Fanuc TP program (LS listing): S103_PK_T13N50.LS

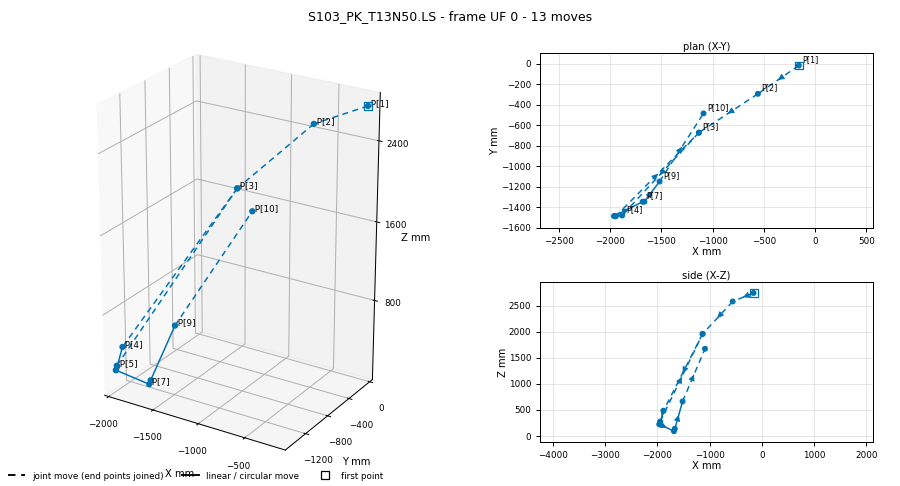
[picture p0: tool path of S103_PK_T13N50.LS in frame UF 0, 13 of 15 moves have a stored position in this frame; points joined in program order, loops and branches not executed]
/PROG  S103_PK_T13N50
/ATTR
OWNER		= MNEDITOR;
COMMENT		= "TL PCK TYP1 N50";
PROG_SIZE	= 4491;
CREATE		= DATE 21-06-09  TIME 06:41:38;
MODIFIED	= DATE 21-06-09  TIME 12:42:18;
FILE_NAME	= S103_PK_;
VERSION		= 0;
LINE_COUNT	= 155;
MEMORY_SIZE	= 4911;
PROTECT		= READ_WRITE;
STORAGE		= SHADOW;
TCD:  STACK_SIZE	= 0,
      TASK_PRIORITY	= 50,
      TIME_SLICE	= 0,
      BUSY_LAMP_OFF	= 0,
      ABORT_REQUEST	= 0,
      PAUSE_REQUEST	= 0;
DEFAULT_GROUP	= 1,*,*,*,*;
CONTROL_CODE	= 00000000 00000000;
/APPL
  HANDLING : TRUE ;
/MN
   1:  !******************************** ;
   2:  ! PATH - PK TOOL FROM N1=STA 70 ;
   3:  !******************************** ;
   4:  !* Robot ID: XXXXXR02B1 ;
   5:  !*    F-19XXXX ;
   6:  !* Line: XXXXXXXX ;
   7:  !* Platform: XX ;
   8:  !* Tool ID: TOOL xx ;
   9:  !* Program: S001_PK_TxxN3_R02 ;
  10:  !* Application: TOOL PICK ;
  11:  !******************************** ;
  12:  ! Author- Esys Automation ;
  13:  !******************************** ;
  14:   ;
  15:  !++++++++++++++++++++++++++++++++ ;
  16:  !ASSIGN PROGRAM PATH VALUES ;
  17:  !-------------------------------- ;
  18:  !Set ATI Tool and World UFrame ;
  19:  UTOOL_NUM=14 ;
  20:  UFRAME_NUM=0 ;
  21:  !++++++++++++++++++++++++++++++++ ;
  22:   ;
  23:  !******************************** ;
  24:  !BEGINNING OF PROGRAM PATH ;
  25:  !MOVE TO NEST 1 TOOL PICK ;
  26:  !******************************** ;
  27:   ;
  28:  !-------------------------------- ;
  29:  LBL[10:MOVE TO TL PICK] ;
  30:   ;
  31:  SET SEGMENT(52) ;
  32:  !SEG(52), Approach Tool Pick ;
  33:   ;
  34:   ;
  35:J P[1] 100% CNT100    ;
  36:J P[2] 100% CNT100    ;
  37:J P[3] 100% CNT100    ;
  38:J P[4] 100% CNT100    ;
  39:   ;
  40:L P[5] 200mm/sec FINE    ;
  41:   ;
  42:L P[6:Pick Tool] 50mm/sec FINE    ;
  43:   ;
  44:  !-------------------------------- ;
  45:  LBL[20:LATCH TOOL] ;
  46:  LATCH TOOL    ;
  47:   ;
  48:  !Add MH Ethernet Device from ;
  49:  !I/O Ethernet table ;
  50:  !which tool has ;
  51:   ;
  52:  !ADD DEVICE ONLINE CALLS ;
  53:  !WITHOUT STATUS CHECK ARG ;
  54:  !FOR ALL EOAT DEVICES ;
  55:  !CALL EN_ONLN(x,y) ;
  56:  !x = EOAT ENET Node # ;
  57:  !y = wait time ;
  58:  CALL EN_ONLN(31,5) ;
  59:  CALL EN_AROFF(31) ;
  60:   ;
  61:  !If TL LCH Pass, Return Home ;
  62:  !If TL LCH Fail, Unlatch TL, ;
  63:  !  MHFault, and Return Home ;
  64:  IF R[170]=1,JMP LBL[30] ;
  65:   ;
  66:  SELECT R[168]=6,JMP LBL[80] ;
  67:         ELSE,JMP LBL[99] ;
  68:   ;
  69:  !-------------------------------- ;
  70:  LBL[30:TOOL CHECK] ;
  71:   ;
  72:  ! Check if Tool Match with PLC ;
  73:  CALL TL_CHK_KM(R[156]) ;
  74:   ;
  75:  !If TL CHK Pass, Return Home ;
  76:  !If TL CHK Fail, Unlatch Tool, ;
  77:  !  MHFault, and Return Home ;
  78:  IF R[170]=1,JMP LBL[40] ;
  79:  IF R[170]=0,JMP LBL[905] ;
  80:   ;
  81:  !-------------------------------- ;
  82:  LBL[40:COMPLETE PATH] ;
  83:  !TL PK COMPLETE. MOVE AWAY ;
  84:  !AND RETURN HOME ;
  85:   ;
  86:  !Set New Tool and World Frame ;
  87:  UTOOL_NUM=2 ;
  88:  UFRAME_NUM=0 ;
  89:   ;
  90:  !Set Payload= Tool ;
  91:  R[221]=2    ;
  92:  PAYLOAD[R[221]] ;
  93:   ;
  94:  SET SEGMENT(53) ;
  95:  !SEG(53), Tool Pick Depart ;
  96:   ;
  97:L P[7] 50mm/sec FINE    ;
  98:L P[8] 1000mm/sec CNT50    ;
  99:L P[9] 1000mm/sec CNT50    ;
 100:   ;
 101:J P[10] 100% CNT100    ;
 102:J P[11] 100% CNT100    ;
 103:   ;
 104:  ! Move To Home ;
 105:  JMP LBL[100] ;
 106:   ;
 107:  !-------------------------------- ;
 108:  LBL[80:LATCHING FAULT] ;
 109:  !MOVE BACK TO HOME WITHOUT TOOL ;
 110:  !on Reverse Path before Tool Pick ;
 111:   ;
 112:  UNLATCH TOOL    ;
 113:   ;
 114:  UFRAME_NUM=0 ;
 115:  UTOOL_NUM=14 ;
 116:   ;
 117:L P[12] 50mm/sec FINE    ;
 118:L P[13] 1000mm/sec CNT50    ;
 119:   ;
 120:J P[14] 100% CNT100    ;
 121:J P[15] 100% CNT100    ;
 122:   ;
 123:   ;
 124:  SET SEGMENT(63) ;
 125:  !SEG(63), Robot Move to Home ;
 126:   ;
 127:  R[132]=0    ;
 128:  GO[71]=0 ;
 129:   ;
 130:  ! Move To Home ;
 131:  JMP LBL[100] ;
 132:   ;
 133:  !-------------------------------- ;
 134:  LBL[99:ABORT PROGRAM] ;
 135:  MESSAGE[...] ;
 136:  MESSAGE[ABORT PROGRAM] ;
 137:  ABORT ;
 138:   ;
 139:  !-------------------------------- ;
 140:  LBL[100:END OF PROGRAM] ;
 141:  END ;
 142:   ;
 143:  !***********FAULTS*********** ;
 144:  LBL[905:Invalid Tool Num] ;
 145:  MESSAGE[...] ;
 146:  MESSAGE[TOOL CHANGER FAULT] ;
 147:  MESSAGE[ ROBOT LATCHED TO] ;
 148:  MESSAGE[ WRONG TOOL.] ;
 149:  MESSAGE[ GI[70] DOES NOT ] ;
 150:  MESSAGE[ MATCH TOOL ID ] ;
 151:  DO[523]=ON ;
 152:  UALM[3] ;
 153:  DO[523]=OFF ;
 154:  JMP LBL[80] ;
 155:   ;
/POS
P[1]{
   GP1:
	UF : 0, UT : 14,		CONFIG : 'N U B, 0, 0, 0',
	X =  -158.400  mm,	Y =   -15.894  mm,	Z =  2741.103  mm,
	W =   -91.792 deg,	P =     -.357 deg,	R =   122.600 deg
};
P[2]{
   GP1:
	UF : 0, UT : 14,		CONFIG : 'N U T, 0, 0, 0',
	X =  -557.806  mm,	Y =  -292.410  mm,	Z =  2577.899  mm,
	W =  -107.925 deg,	P =    -3.536 deg,	R =   122.979 deg
};
P[3]{
   GP1:
	UF : 0, UT : 14,		CONFIG : 'N U T, 0, 0, 0',
	X = -1134.710  mm,	Y =  -671.782  mm,	Z =  1955.941  mm,
	W =  -117.901 deg,	P =    -3.388 deg,	R =   113.635 deg
};
P[4:""]{
   GP1:
	UF : 0, UT : 14,		CONFIG : 'N U T, 0, 0, 0',
	X = -1884.319  mm,	Y = -1480.761  mm,	Z =   484.909  mm,
	W =  -160.186 deg,	P =     -.015 deg,	R =    91.377 deg
};
P[5]{
   GP1:
	UF : 0, UT : 14,		CONFIG : 'N U T, 0, 0, 0',
	X = -1946.275  mm,	Y = -1485.539  mm,	Z =   267.115  mm,
	W =  -160.189 deg,	P =      .120 deg,	R =    91.629 deg
};
P[6:"Pick Tool"]{
   GP1:
	UF : 0, UT : 14,		CONFIG : 'N U T, 0, 0, 0',
	X = -1961.425  mm,	Y = -1486.060  mm,	Z =   225.038  mm,
	W =  -160.189 deg,	P =      .120 deg,	R =    91.629 deg
};
P[7]{
   GP1:
	UF : 0, UT : 2,		CONFIG : 'N U T, 0, 0, 0',
	X = -1683.492  mm,	Y = -1346.337  mm,	Z =    92.333  mm,
	W =  -161.730 deg,	P =      .342 deg,	R =    89.831 deg
};
P[8]{
   GP1:
	UF : 0, UT : 2,		CONFIG : 'N U T, 0, 0, 0',
	X = -1666.820  mm,	Y = -1346.000  mm,	Z =   138.620  mm,
	W =  -161.730 deg,	P =      .342 deg,	R =    89.831 deg
};
P[9]{
   GP1:
	UF : 0, UT : 2,		CONFIG : 'N U T, 0, 0, 0',
	X = -1518.219  mm,	Y = -1148.677  mm,	Z =   662.684  mm,
	W =  -149.064 deg,	P =     3.941 deg,	R =    99.038 deg
};
P[10]{
   GP1:
	UF : 0, UT : 2,		CONFIG : 'N U T, 0, 0, 0',
	X = -1089.020  mm,	Y =  -483.560  mm,	Z =  1671.146  mm,
	W =  -119.401 deg,	P =    -2.194 deg,	R =   112.860 deg
};
P[11]{
   GP1:
	UF : 0, UT : 2,
	J1=  -145.477 deg,	J2=   -28.708 deg,	J3=    89.000 deg,
	J4=     2.573 deg,	J5=   -83.800 deg,	J6=   -90.000 deg
};
P[12]{
   GP1:
	UF : 0, UT : 14,		CONFIG : 'N U T, 0, 0, 0',
	X = -1961.425  mm,	Y = -1486.060  mm,	Z =   225.038  mm,
	W =  -160.189 deg,	P =      .120 deg,	R =    91.629 deg
};
P[13]{
   GP1:
	UF : 0, UT : 14,		CONFIG : 'N U T, 0, 0, 0',
	X = -1948.077  mm,	Y = -1489.017  mm,	Z =   276.693  mm,
	W =  -160.188 deg,	P =     -.018 deg,	R =    91.207 deg
};
P[14]{
   GP1:
	UF : 0, UT : 14,		CONFIG : 'N U T, 0, 0, 0',
	X = -1134.710  mm,	Y =  -671.782  mm,	Z =  1955.941  mm,
	W =  -117.901 deg,	P =    -3.388 deg,	R =   113.635 deg
};
P[15]{
   GP1:
	UF : 0, UT : 14,
	J1=  -145.476 deg,	J2=   -28.707 deg,	J3=    89.000 deg,
	J4=     2.574 deg,	J5=   -83.800 deg,	J6=   -90.001 deg
};
/END
